FUNCTION_BLOCK FB_CSVPersistentEventStorage IMPLEMENTS I_PersistentEventStorage
VAR
	eWriteState : (File_Open_Trigger,File_Open,Wait_For_Event,Write_Event_Trigger,Write_Event,File_Close_Trigger,File_Close,Error);
	fbFileOpen:FB_FileOpen:= (sPathName:= 'C:\Users\Beckhoff\Desktop\Event.log',nMode:=FOPEN_MODEAPPEND OR FOPEN_MODETEXT);
	fbFilePuts: FB_FilePuts;
//	fbFileWrite:FB_FileWrite;
	fbFileClose:FB_FileClose;
	stEventWrittenToFile:ST_Event;
	CSVString:T_MaxString;
END_VAR

CASE eWriteState OF
	File_Open_Trigger:
		fbFileOpen(bExecute:=TRUE);
		eWriteState:=File_Open;
		
	File_Open:
		fbFileOpen(bExecute:=FALSE);
		IF fbFileOpen.bError THEN
			eWriteState:=Error;
		ELSIF NOT fbFileOpen.bBusy AND fbFileOpen.hFile<>0 THEN
			eWriteState:=Wait_For_Event;
		END_IF;
		
	Wait_For_Event:
	//do nothing
	
	Write_Event_Trigger:
		CSVString:=CreateCSVString(stEvent:=stEventWrittenToFile);
		fbFilePuts(bExecute:=TRUE,sLine:=CSVString,hFile:=fbFileOpen.hFile);
		eWriteState:=Write_Event;	

	Write_Event:
		fbFilePuts(bExecute:=FALSE);
		IF fbFilePuts.bError THEN
			eWriteState:=Error;
		ELSIF NOT fbFilePuts.bBusy THEN
			eWriteState:=File_Close_Trigger;
		END_IF;
	File_Close_Trigger:
		fbFileClose(bExecute:=TRUE,hFile:=fbFileOpen.hFile);
		eWriteState:=File_Close;	
	File_Close:
		fbFileClose(bExecute:=FALSE);
		IF fbFileClose.bError THEN
			eWriteState:=Error;
		ELSIF NOT fbFileClose.bBusy THEN
			eWriteState:=File_Open_Trigger;
		END_IF;	
END_CASE;

METHOD PRIVATE CreateCSVString : T_MaxString
VAR_INPUT
	stEvent : REFERENCE TO ST_Event;
END_VAR
VAR
	TempString : T_MaxString;
END_VAR

TempString:= TO_STRING(stEvent.eEventTypes);
TempString:=Concat(STR1:= TempString,STR2:=',');
TempString:=Concat(STR1:= TempString,STR2:=TO_STRING(stEvent.eEventSeverity));
TempString:=Concat(STR1:= TempString,STR2:=',');
TempString:=Concat(STR1:= TempString,STR2:=TO_STRING(stEvent.eEventIdentity));
TempString:=Concat(STR1:= TempString,STR2:=',');
TempString:=Concat(STR1:= TempString,STR2:=stEvent.eEventText);
TempString:=Concat(STR1:= TempString,STR2:=',');
TempString:=Concat(STR1:= TempString,STR2:=TO_STRING(stEvent.dtTimestamp));
TempString:=Concat(STR1:= TempString,STR2:='$N');

CreateCSVString:=TempString;
END_METHOD

{warning 'add method implementation '}
METHOD StoreEvent
VAR_INPUT
	stEvent	: ST_Event;
END_VAR
//write csv code
IF eWriteState=Wait_For_Event THEN
	stEventWrittenToFile:=stEvent;
	eWriteState:= Write_Event_Trigger;
END_IF
END_METHOD

END_FUNCTION_BLOCK

(* stored: Version 1.1.0.1, ProductVersion 3.1.4024.12
   POU FB_CSVPersistentEventStorage: Id {f7618ef2-831b-4fb5-bf06-e736f4bd9e12}, SpecialFunc None
   Method CreateCSVString: Id {13de78ee-0463-440c-9a6c-aff8a9fbc1d2}
   Method StoreEvent: Id {4653cad3-d932-4e8e-a7ca-8a5cbd78a6a2} *)
